TYPE ST_SMSDataSetEntry_Read :
STRUCT
	Message : STRING(160);  // Commande envoyé par message
	Num		: STRING(20);  //  Numéro de l'utilisateur
END_STRUCT
END_TYPE

(* stored: Version 1.1.0.1, ProductVersion 3.1.4024.6
   DUT ST_SMSDataSetEntry_Read: Id {2ef04086-c2e9-4ce9-ba07-b36c18a487ee} *)
